(* IEC 61131-3 sources: WaterIrrigation/Virtual Sim PLC Package/build, 2 files *)

(* ---- plc.st ---- *)
TYPE
  LOGLEVEL : (CRITICAL, WARNING, INFO, DEBUG) := INFO;
END_TYPE

FUNCTION_BLOCK LOGGER
  VAR_INPUT
    TRIG : BOOL;
    MSG : STRING;
    LEVEL : LOGLEVEL := INFO;
  END_VAR
  VAR
    TRIG0 : BOOL;
  END_VAR

  IF TRIG AND NOT TRIG0 THEN
  {{
   LogMessage(GetFbVar(LEVEL),(char*)GetFbVar(MSG, .body),GetFbVar(MSG, .len));
  }}
  END_IF;
  TRIG0:=TRIG;
END_FUNCTION_BLOCK

FUNCTION_BLOCK python_eval
  VAR_INPUT
    TRIG : BOOL;
    CODE : STRING;
  END_VAR
  VAR_OUTPUT
    ACK : BOOL;
    RESULT : STRING;
  END_VAR
  VAR
    STATE : DWORD;
    BUFFER : STRING;
    PREBUFFER : STRING;
    TRIGM1 : BOOL;
    TRIGGED : BOOL;
  END_VAR

  {extern void __PythonEvalFB(int, PYTHON_EVAL*);__PythonEvalFB(0, data__);}
END_FUNCTION_BLOCK

FUNCTION_BLOCK python_poll
  VAR_INPUT
    TRIG : BOOL;
    CODE : STRING;
  END_VAR
  VAR_OUTPUT
    ACK : BOOL;
    RESULT : STRING;
  END_VAR
  VAR
    STATE : DWORD;
    BUFFER : STRING;
    PREBUFFER : STRING;
    TRIGM1 : BOOL;
    TRIGGED : BOOL;
  END_VAR

  {extern void __PythonEvalFB(int, PYTHON_EVAL*);__PythonEvalFB(1,(PYTHON_EVAL*)(void*)data__);}
END_FUNCTION_BLOCK

FUNCTION_BLOCK python_gear
  VAR_INPUT
    N : UINT;
    TRIG : BOOL;
    CODE : STRING;
  END_VAR
  VAR_OUTPUT
    ACK : BOOL;
    RESULT : STRING;
  END_VAR
  VAR
    py_eval : python_eval;
    COUNTER : UINT;
    _TMP_ADD10_OUT : UINT;
    _TMP_EQ13_OUT : BOOL;
    _TMP_SEL15_OUT : UINT;
    _TMP_AND7_OUT : BOOL;
  END_VAR

  _TMP_ADD10_OUT := ADD(COUNTER, 1);
  _TMP_EQ13_OUT := EQ(N, _TMP_ADD10_OUT);
  _TMP_SEL15_OUT := SEL(_TMP_EQ13_OUT, _TMP_ADD10_OUT, 0);
  COUNTER := _TMP_SEL15_OUT;
  _TMP_AND7_OUT := AND(_TMP_EQ13_OUT, TRIG);
  py_eval(TRIG := _TMP_AND7_OUT, CODE := CODE);
  ACK := py_eval.ACK;
  RESULT := py_eval.RESULT;
END_FUNCTION_BLOCK

PROGRAM WaterIrrigation
  VAR
    OUTGOING_VALVE : BOOL;
    OUTGOING_PUMP : BOOL;
    INCOMING_PUMP : BOOL;
    TANK_FULL : BOOL;
    PULSE : BOOL;
    TANK_EMPTY : BOOL;
    MANUAL : BOOL;
    PB_INCOMING_OPEN : BOOL;
    PB_INCOMING_CLOSE : BOOL;
    PB_OUTGOING_OPEN : BOOL;
    PB_OUTGOING_CLOSE : BOOL;
    MAX_TANK_LEVEL : INT := 10;
    TANK_LEVEL_VALUE : INT := 10;
    WATER_MOISTURE : INT := 10;
  END_VAR
  VAR
    TON0 : TON;
    TOF0 : TOF;
    CTUD0 : CTUD;
    R_TRIG1 : R_TRIG;
    R_TRIG2 : R_TRIG;
  END_VAR

  OUTGOING_PUMP := OUTGOING_VALVE;
  R_TRIG1(CLK := PULSE AND INCOMING_PUMP);
  R_TRIG2(CLK := PULSE AND OUTGOING_PUMP);
  CTUD0(CU := R_TRIG1.Q, CD := R_TRIG2.Q, PV := MAX_TANK_LEVEL);
  TANK_FULL := CTUD0.QU;
  TANK_EMPTY := CTUD0.QD;
  TANK_LEVEL_VALUE := CTUD0.CV;
  TON0(IN := NOT(PULSE), PT := T#500ms);
  TOF0(IN := TON0.Q, PT := T#500ms);
  PULSE := TOF0.Q;
  INCOMING_PUMP := PB_INCOMING_CLOSE AND (INCOMING_PUMP OR NOT(PB_INCOMING_OPEN));
  OUTGOING_VALVE := NOT(PB_OUTGOING_CLOSE) AND (OUTGOING_VALVE OR PB_OUTGOING_OPEN);
END_PROGRAM

CONFIGURATION Config0

  RESOURCE Res0 ON PLC
    TASK task0(INTERVAL := T#20ms,PRIORITY := 0);
    PROGRAM instance0 WITH task0 : WaterIrrigation;
  END_RESOURCE
END_CONFIGURATION

(* ---- generated_plc.st ---- *)
PROGRAM WaterIrrigation
  VAR
    OUTGOING_VALVE AT %QX0.0 : BOOL;
    OUTGOING_PUMP AT %QX0.1 : BOOL;
    INCOMING_PUMP AT %QX0.2 : BOOL;
    TANK_FULL AT %QX0.3 : BOOL;
    PULSE AT %QX0.4 : BOOL;
    TANK_EMPTY AT %QX0.5 : BOOL;
    MANUAL AT %QX0.6 : BOOL;
    PB_INCOMING_OPEN AT %IX0.0 : BOOL;
    PB_INCOMING_CLOSE AT %IX0.1 : BOOL;
    PB_OUTGOING_OPEN AT %IX0.2 : BOOL;
    PB_OUTGOING_CLOSE AT %IX0.3 : BOOL;
    MAX_TANK_LEVEL AT %QW0 : INT := 10;
    TANK_LEVEL_VALUE AT %QW2 : INT := 10;
    WATER_MOISTURE AT %QW3 : INT := 10;
  END_VAR
  VAR
    TON0 : TON;
    TOF0 : TOF;
    CTUD0 : CTUD;
    R_TRIG1 : R_TRIG;
    R_TRIG2 : R_TRIG;
  END_VAR

  OUTGOING_PUMP := OUTGOING_VALVE;
  R_TRIG1(CLK := PULSE AND INCOMING_PUMP);
  R_TRIG2(CLK := PULSE AND OUTGOING_PUMP);
  CTUD0(CU := R_TRIG1.Q, CD := R_TRIG2.Q, PV := MAX_TANK_LEVEL);
  TANK_FULL := CTUD0.QU;
  TANK_EMPTY := CTUD0.QD;
  TANK_LEVEL_VALUE := CTUD0.CV;
  TON0(IN := NOT(PULSE), PT := T#500ms);
  TOF0(IN := TON0.Q, PT := T#500ms);
  PULSE := TOF0.Q;
  INCOMING_PUMP := PB_INCOMING_CLOSE AND (INCOMING_PUMP OR NOT(PB_INCOMING_OPEN));
  OUTGOING_VALVE := NOT(PB_OUTGOING_CLOSE) AND (OUTGOING_VALVE OR PB_OUTGOING_OPEN);
END_PROGRAM

CONFIGURATION Config0

  RESOURCE Res0 ON PLC
    TASK task0(INTERVAL := T#20ms,PRIORITY := 0);
    PROGRAM instance0 WITH task0 : WaterIrrigation;
  END_RESOURCE
END_CONFIGURATION
